// LS Electric XG5000 project: XGK256S
// PLC LSPLC

PROGRAM NewProgram (task: 스캔 프로그램)

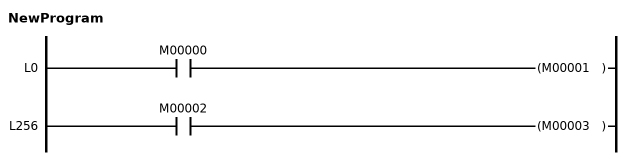
; L0
LOAD      M00000
OUT       M00001
; L256
LOAD      M00002
OUT       M00003